{attribute 'linkalways'} 
{attribute 'no_explicit_call' := 'This FB is a CLASS and must be accessed using methods or properties'}
{attribute 'enable_dynamic_creation'}
FUNCTION_BLOCK Node_F_VN_HuMomentInvariants EXTENDS VisionNode
VAR
    stMoments : _TcVnMoments;
    aHuInvariants : _TcVnArray7_LREAL;
    hrPrev : _HRESULT(S_OK);
	hresult : _HRESULT(S_OK);
END_VAR

METHOD PUBLIC  Clone : I_Node
VAR
	pNode : POINTER TO Node_F_VN_HuMomentInvariants;
END_VAR
pNode := __NEW(Node_F_VN_HuMomentInvariants);
Clone := pNode^;
END_METHOD

METHOD FB_init : BOOL
VAR_INPUT
	bInitRetains : BOOL; // if TRUE, the retain variables are initialized (warm start / cold start)
	bInCopyCode : BOOL;  // if TRUE, the instance afterwards gets moved into the copy code (online change)
END_VAR
AddInput('stMoments', stMoments);
AddInput('hrPrev', hrPrev);
AddOutput('aHuInvariants', aHuInvariants);
AddOutput('hresult',hresult);
END_METHOD

METHOD PROTECTED  OnExecute : HRESULT
hresult.Value := F_VN_HuMomentInvariants(
	stMoments := stMoments.Value,
    aHuInvariants := aHuInvariants.Value,
	hrPrev:= hrPrev.Value);
END_METHOD

METHOD PUBLIC PreExecutionCheck
VAR_INPUT
	Check : I_PreExecutionChecks;
END_VAR
END_METHOD

END_FUNCTION_BLOCK

(* stored: Version 1.1.0.1, ProductVersion 3.1.4024.13
   POU Node_F_VN_HuMomentInvariants: Id {8d96b3fc-ba79-070d-05d9-8b6c15bcec97}, SpecialFunc None
   Folder Constructor: Id {176a5d38-5389-0573-2346-3096ead23911}
   Method Clone: Id {4bd8c3e3-cfb6-057e-3385-018159bade73}
   Method FB_init: Id {e1072ac9-0a49-02a4-3b05-88cba79681f1}
   Method OnExecute: Id {51d69cb4-f15b-05fc-3228-7a7d89cf83ed}
   Method PreExecutionCheck: Id {1a280466-5c27-0ea5-2f2c-679adf1817ab} *)
